PROGRAM MAIN
VAR
	i : INT;
END_VAR

i := i+1;

END_PROGRAM

(* stored: Version 1.1.0.1, ProductVersion 3.1.4024.12
   POU MAIN: Id {71cdf35c-f4d4-40cc-9bda-d1b442d54f21}, SpecialFunc None *)
